(* PLC project demo-project, Synthetic Demo Industrial XML Fingerprint *)

PROGRAM DemoProgram

Counter := Counter + 1;
END_PROGRAM
